FUNCTION_BLOCK FB_VarByteBuffer EXTENDS FB_VarByteBufferBase IMPLEMENTS I_VarByteBuffer
VAR
END_VAR

METHOD Push : BOOL
VAR_INPUT
	pData : pvoid;
	cbSize : UDINT;
END_VAR
VAR;
	res			: UDINT;
END_VAR
IF (THIS^._pBuffer = 0) OR (THIS^._nCapacity = 0) THEN RETURN; END_IF;		// Check initialization
IF pData = 0 THEN RETURN; END_IF											// Check input
IF THIS^.FreeBytes < cbSize THEN RETURN; END_IF;

res := memcpy(THIS^._pBuffer + THIS^._nHead,pData,cbSize);
IF res <> cbSize THEN
	THIS^._nError := THIS^._nError + 1; 
	RETURN;
END_IF

THIS^._nHead := THIS^._nHead + cbSize;

Push := TRUE;
END_METHOD

END_FUNCTION_BLOCK

(* stored: Version 1.1.0.1
   POU FB_VarByteBuffer: Id {4e19349b-1227-46f1-97cb-14d3a766e6ec}, SpecialFunc None
   Method Push: Id {e4bd66c9-d210-422e-b417-2a1820ac5d79} *)
